TYPE ST_Event :
STRUCT
	eEventType		: E_EventType;
	eSeverity 		: E_Severity := E_Severity.Event;
	sMessage	 	: STRING(255);
	dTimestamp 		: DATE_AND_TIME;
END_STRUCT
END_TYPE

(* stored: Version 1.1.0.1
   DUT ST_Event: Id {493c11c6-cf57-4007-9b07-d443ab2430c6} *)
